(* IEC 61131-3 sources: programs/VI-54/VI-54_20171205/VI-54_20171205/Stations/Screen/LseClass170718/Class/ReceptBase, 1 file *)

(* ---- ReceptBase.st ---- *)
(*!
<Class
	Name               = "ReceptBase"
	Revision           = "0.0"
	RealtimeTask       = "false"
	CyclicTask         = "false"
	BackgroundTask     = "false"
	Sigmatek           = "false"
	OSInterface        = "false"
	HighPriority       = "false"
	Automatic          = "false"
	UpdateMode         = "Prescan"
	SharedCommandTable = "true"
	Objectsize         = "(284,120)">
	<Channels>
		<Server Name="Refresh" Visualized="false" Initialize="false" WriteProtected="false" Retentive="false"/>
		<Server Name="Size" Visualized="false" Initialize="false" WriteProtected="true" Retentive="false"/>
		<Client Name="Data" Required="true" Internal="false"/>
	</Channels>
</Class>
*)
ReceptBase : CLASS
  //Servers:
	Refresh 	: SvrChCmd_DINT;
	Size 	: SvrCh_DINT;
  //Clients:
	Data 	: CltChCmd_MerkerEx;
  //Variables:
		ReceptPtr 	: ^DataRecipeStr;
  //Functions:

	FUNCTION VIRTUAL GLOBAL Init;

	FUNCTION VIRTUAL GLOBAL DefaultPara;

	FUNCTION VIRTUAL GLOBAL RefreshPara;

	FUNCTION VIRTUAL GLOBAL Refresh::Write
		VAR_INPUT
			input (EAX) 	: DINT;
		END_VAR
		VAR_OUTPUT
			result (EAX) 	: DINT;
		END_VAR;
  //Tables:
	FUNCTION @STD
		VAR_OUTPUT
			ret_code	: CONFSTATES;
		END_VAR;
	FUNCTION GLOBAL TAB @CT_;
END_CLASS;

#pragma usingLtd MerkerEx

FUNCTION VIRTUAL GLOBAL ReceptBase::Init

  // Set data size
  if Data.GetSize() <> sizeof(DataRecipeStr) then
    Data.SetSize(udSize:= sizeof(DataRecipeStr));
  end_if;

  // Get pointer
  if _FirstScan = 1 then
    ReceptPtr$^Usint := Data.GetDataPtr();
    if ReceptPtr$^Usint = Data.GetDataPtr() then
      RefreshPara();
    end_if;
  end_if;

END_FUNCTION

FUNCTION VIRTUAL GLOBAL ReceptBase::DefaultPara

END_FUNCTION

FUNCTION VIRTUAL GLOBAL ReceptBase::RefreshPara

END_FUNCTION

FUNCTION VIRTUAL GLOBAL ReceptBase::Refresh::Write
	VAR_INPUT
		input (EAX) 	: DINT;
	END_VAR
	VAR_OUTPUT
		result (EAX) 	: DINT;
	END_VAR

  Refresh := input;
  if ReceptPtr <> 0 then
    RefreshPara();
  end_if;
 	result := Refresh;

END_FUNCTION
